FUNCTION_BLOCK fbLightControl_ButtonAndDetect
		
VAR_INPUT
	bButton				: BOOL;
	bDeurDetectie		: BOOL;
	bForceOff			: BOOL;
	bForceOn			: BOOL;
	bDetection			: BOOL;
	bInhibit			:BOOL;
	
	//tInhibitTime		:TIME := T#60s;
    tDeurOpenTime		:TIME := T#10m;
END_VAR
VAR_OUTPUT
	bLight				: BOOL;
	
END_VAR
VAR
	InputTrigger		: R_trig; 
	DetectieTrigger		: R_trig; 
	DeurTrigger			: R_trig; 
	//TimerInhibit		: TOF; 
	TimerDeurdetectie	: TON;
	bInternLichtVarKnop : BOOL;
	bOverneemDeurDetectie :BOOL;
	
END_VAR

// This is the first version, ignoring all debounce timers and other issues 
// Base function is a to allow switching a light on and of and having a general reset and general on ( used for construcion)

//Button detection
InputTrigger(CLK :=  bButton);

//rising edge detection used for the optical detection and deur detection
DetectieTrigger(clk := bDetection);
DeurTrigger(clk := bDeurDetectie);
// button function
IF InputTrigger.Q THEN
	
	IF bInternLichtVarKnop OR bOverneemDeurDetectie THEN
		bOverneemDeurDetectie :=  FALSE;
	END_IF
	bInternLichtVarKnop := NOT(bInternLichtVarKnop);

END_IF

// Dit onderdeel triggert als de deur opent en blijft de ingestelde tijd lopen na het sleuiten

IF DetectieTrigger.Q OR DeurTrigger.Q THEN 
	bOverneemDeurDetectie := TRUE;
END_IF

TimerDeurdetectie(In := bOverneemDeurDetectie AND(NOT(DetectieTrigger.Q )), PT:= tDeurOpenTime);


IF TimerDeurdetectie.Q THEN
	bOverneemDeurDetectie := FALSE;
END_IF

// Deze functie zorgt voor alles aan/Uit Functionaliteit
IF bForceOff THEN
	bInternLichtVarKnop := FALSE;
	bOverneemDeurDetectie := FALSE;
END_IF

IF bForceOn THEN
	bInternLichtVarKnop := TRUE;
END_IF


bLight := (bInternLichtVarKnop OR  bOverneemDeurDetectie) ;




(*function notes: long klick functionality not added, most likley this will be part of another function
This could be a dedicated filter function linked to these functions as needed
*)

END_FUNCTION_BLOCK

(* stored: Version 1.1.0.1, ProductVersion 3.1.4024.12
   POU fbLightControl_ButtonAndDetect: Id {4ce95e57-7aca-434a-866b-1258781c6cb7}, SpecialFunc None *)
